Yaskawa INFORM job: FRONT_SEARCH_0ST-2_5040.JBI

/JOB
//NAME FRONT_SEARCH_0ST-2_5040
///FOLDERNAME 02-SKRZYNIE_JOBS
//POS
///NPOS 102,102,0,15,0,0
///TOOL 0
///POSTYPE PULSE
///PULSE
C00000=0,-52280,40443,0,-64237,0
C00001=0,-44333,40442,1,-36510,2
C00002=0,-77502,-19682,2,-20075,2
C00003=-31499,-58302,-23356,15027,12889,-13082
C00004=-52768,-43016,-26078,18373,38595,-18774
C00005=-77982,-19483,-4354,30116,56383,-30765
C00006=-53036,-11528,-12218,12363,64665,-17409
C00007=-53036,-11528,-12218,12363,64665,-17409
C00008=-51536,-9474,-10276,11905,64649,-16876
C00009=-51739,-9114,-7787,12104,63269,-17104
C00010=-53036,-11528,-12218,12363,64665,-17409
C00011=-17541,-26226,-24397,927,59032,-5038
C00012=-17541,-26226,-24397,927,59032,-5038
C00013=-16950,-23991,-22741,715,59568,-4818
C00014=-17036,-23563,-20101,755,58071,-4857
C00015=-17541,-26226,-24397,927,59032,-5038
C00016=34102,-23192,-21614,-15638,64271,13209
C00017=33423,-21885,-20599,-15423,64418,12942
C00018=32426,-19856,-18975,-15106,64629,12551
C00019=32578,-19611,-17013,-15290,63535,12762
C00020=33423,-21885,-20599,-15423,64418,12942
C00021=59339,-6070,-6417,-20979,72191,20891
C00022=59339,-6070,-6417,-20979,72191,20891
C00023=57897,-4256,-4562,-20702,71913,20431
C00024=58108,-3992,-2506,-20878,70835,20713
C00025=59339,-6070,-6417,-20979,72191,20891
C00026=42744,-35904,-30225,-18322,62562,16651
C00027=-53036,-11528,-12218,12363,64665,-17409
C00028=-77982,-26538,-29134,27151,66629,-27745
C00029=-70983,-8594,-1966,26503,59809,-49670
C00030=-80152,19776,40785,37351,72704,-50428
C00031=-79984,20154,42529,37516,71911,-50638
C00032=-79233,18397,40079,37458,71885,-50340
C00033=-79984,20154,42529,37516,71911,-50638
C00034=-73519,23289,38838,28890,77081,-45618
C00035=-73519,24511,42682,29072,75582,-46027
C00036=-73519,23289,38838,28890,77081,-45618
C00037=-88897,15706,42282,50101,71325,-56974
C00038=-88897,15706,42282,50101,71325,-56974
C00039=-87612,12343,37838,50071,70996,-56519
C00040=-85283,14202,40272,50301,69633,-56165
C00041=-87338,12550,38107,50098,70839,-56476
C00042=-84952,-1789,13569,34660,47724,-58955
C00043=-67641,-1674,11109,10330,44856,-44725
C00044=-66443,961,13975,9688,44721,-44210
C00045=-67641,-1674,11109,10330,44856,-44725
C00046=-67641,-376,15347,10694,42950,-44967
C00047=-67641,-1674,11109,10330,44856,-44725
C00048=-79040,417,20398,15965,28992,-57786
C00049=-76655,5212,30978,15501,25024,-57306
C00050=-76655,6949,35816,16758,23084,-57955
C00051=-76655,5212,30978,15501,25024,-57306
C00052=-74761,6919,33010,13466,24593,-56049
C00053=-80460,-2874,12270,15804,32253,-57809
C00054=-61258,-29124,-13156,26560,43617,-22150
C00055=-30420,-40507,-29240,27153,53235,15188
C00056=-18589,-38725,-21450,23338,47896,18931
C00057=-17722,-35233,-16455,23322,46926,19051
C00058=-17722,-33749,-12435,23948,45421,18620
C00059=-17722,-33892,-12819,23887,45564,18661
C00060=-16677,-31133,-11209,23138,46167,19311
C00061=-17819,-35820,-17540,23246,47228,19090
C00062=-74104,-11494,-6266,31916,75042,4269
C00063=-71226,-7329,2631,32115,71468,4273
C00064=-71226,-6504,5446,32343,70365,3922
C00065=-71226,-6611,5086,32313,70505,3967
C00066=-68386,-4058,7675,32040,69573,4789
C00067=-73314,-9412,-353,32206,72648,3829
C00068=51751,-31069,-22965,-10739,49070,48663
C00069=49028,-23852,-11575,-9841,46366,47823
C00070=49028,-23004,-8935,-10039,45204,47956
C00071=49028,-23118,-9286,-10013,45357,47939
C00072=47000,-20813,-7527,-8928,45644,47024
C00073=50476,-26208,-15307,-10408,47325,48332
C00074=90602,-5375,6902,-38786,69848,59444
C00075=83174,19950,50269,-44999,67580,58220
C00076=82362,17902,47383,-44926,67511,57879
C00077=83515,19072,48341,-44798,68200,58056
C00078=78091,19382,40247,-36371,72286,52960
C00079=78091,20664,44011,-36670,70997,53443
C00080=78091,19382,40247,-36371,72286,52960
C00081=88699,7296,38566,-55615,63182,60372
C00082=86803,3068,32674,-55410,62638,59657
C00083=84852,4315,34115,-55564,61561,59330
C00084=86803,3068,32674,-55410,62638,59657
C00085=92770,-2803,21719,-53893,67577,59421
C00086=73393,-10627,10934,-27897,30744,62458
C00087=70789,-6606,18800,-27824,27830,62140
C00088=69654,-4593,20814,-26755,27596,61444
C00089=70789,-6606,18800,-27824,27830,62140
C00090=70789,-5070,23059,-29482,26284,63017
C00091=70789,-6606,18800,-27824,27830,62140
C00092=83486,-8736,6503,-27040,35338,66550
C00093=77831,-2041,26192,-25270,18452,68895
C00094=77967,1961,32070,-26860,17569,69698
C00095=77967,5243,40752,-32914,14549,72656
C00096=77967,1961,32070,-26860,17569,69698
C00097=74560,4730,35257,-21622,16551,66717
C00098=77967,1961,32070,-26860,17569,69698
C00099=81109,-22356,2664,-22493,33121,60116
C00100=86168,-49730,-13668,-23926,46819,49343
C00101=44183,-52048,-7537,-24795,46064,51426
BC00000=868944
BC00001=857186
BC00002=897097
BC00003=897097
BC00004=897097
BC00005=897097
BC00006=912458
BC00007=912458
BC00008=912458
BC00009=912458
BC00010=912458
BC00011=912458
BC00012=912458
BC00013=912458
BC00014=912458
BC00015=912458
BC00016=912458
BC00017=912458
BC00018=912458
BC00019=912458
BC00020=912458
BC00021=912458
BC00022=912458
BC00023=912458
BC00024=912458
BC00025=912458
BC00026=912458
BC00027=912458
BC00028=912458
BC00029=912458
BC00030=912458
BC00031=912460
BC00032=912460
BC00033=912460
BC00034=912460
BC00035=912460
BC00036=912460
BC00037=912460
BC00038=912460
BC00039=912460
BC00040=912460
BC00041=912460
BC00042=912460
BC00043=912460
BC00044=912460
BC00045=912460
BC00046=912460
BC00047=912460
BC00048=912460
BC00049=912460
BC00050=912460
BC00051=912460
BC00052=912460
BC00053=912460
BC00054=912461
BC00055=912462
BC00056=912462
BC00057=912462
BC00058=912462
BC00059=912462
BC00060=912462
BC00061=912462
BC00062=912462
BC00063=912462
BC00064=912462
BC00065=912462
BC00066=912434
BC00067=912448
BC00068=912448
BC00069=912448
BC00070=912448
BC00071=912448
BC00072=912448
BC00073=912448
BC00074=912462
BC00075=912462
BC00076=912462
BC00077=912462
BC00078=912462
BC00079=912462
BC00080=912462
BC00081=912462
BC00082=912462
BC00083=912462
BC00084=912462
BC00085=912462
BC00086=912462
BC00087=912462
BC00088=912462
BC00089=912462
BC00090=912462
BC00091=912462
BC00092=912462
BC00093=912462
BC00094=912462
BC00095=912462
BC00096=912462
BC00097=912462
BC00098=912462
BC00099=880677
BC00100=854232
BC00101=807451
///POSTYPE BASE
///RECTAN
///RCONF 1,0,0,0,0,0,0,0,0,0,0,0,0,0,0,0,0,0,0,0,0,0,0,0
P00006=0.000,0.000,0.000,0.0000,0.0000,0.0000
///RCONF 0,0,0,0,0,0,0,0,0,0,0,0,0,0,0,0,0,0,0,0,0,0,0,0
P00058=0.000,0.000,3.000,0.0000,0.0000,0.0000
P00350=11.519,-0.008,1.149,0.0000,0.0000,0.0000
P00351=13.563,-0.027,-0.653,0.0000,0.0000,0.0000
P00352=13.252,-0.027,-0.827,0.0000,0.0000,0.0000
P00353=10.971,-0.082,0.776,0.0000,0.0000,0.0000
P00399=-2.449,0.031,8.825,0.0000,0.0000,0.0000
P00400=5.920,-3.503,-0.024,0.0000,0.0000,0.0000
P00401=3.430,-0.021,1.131,0.0000,0.0000,0.0000
P00402=-0.253,1.107,3.062,0.0000,0.0000,0.0000
P00403=-3.666,-0.015,5.328,0.0000,0.0000,0.0000
P00405=2.420,0.007,1.427,0.0000,0.0000,0.0000
P00406=3.513,-0.022,0.429,0.0000,0.0000,0.0000
P00415=-1.781,-1.303,3.250,0.0000,0.0000,0.0000
P00416=0.027,1.119,3.078,0.0000,0.0000,0.0000
//INST
///DATE 2024/05/14 19:22
///ATTR SC,RW
///GROUP1 RB1,BS1
NOP
MOVJ C00000 BC00000 VJ=10.00
MOVJ C00001 BC00001 VJ=30.00
MOVJ C00002 BC00002 VJ=20.00
MOVJ C00003 BC00003 VJ=20.00
MOVJ C00004 BC00004 VJ=20.00
MOVJ C00005 BC00005 VJ=10.00
'DODANE
'SZUKANIE FRONT
'------------------------
'503
'------------------------
MOVL C00006 BC00006 V=166.7
MOVL C00007 BC00007 V=66.7 PL=0
REFP 3 C00008 BC00008
CALL JOB:SEARCH-R1
IMOV P0058 V=16.7
SET P0350 P0006
SFTON P0350
REFP 3 C00009 BC00009
CALL JOB:SEARCH-R1
SET P0350 P0006
SFTON P0350
MOVL C00010 BC00010 V=66.7 PL=0
SFTOF
'------------------------
'------------------------
'502
'------------------------
MOVL C00011 BC00011 V=166.7
MOVL C00012 BC00012 V=66.7 PL=0
REFP 3 C00013 BC00013
CALL JOB:SEARCH-R1
IMOV P0058 V=16.7
SET P0351 P0006
SFTON P0351
REFP 3 C00014 BC00014
CALL JOB:SEARCH-R1
SET P0351 P0006
SFTON P0351
MOVL C00015 BC00015 V=66.7 PL=0
SFTOF
'------------------------
'------------------------
'501
'------------------------
MOVL C00016 BC00016 V=166.7
MOVL C00017 BC00017 V=66.7 PL=0
REFP 3 C00018 BC00018
CALL JOB:SEARCH-R1
IMOV P0058 V=16.7
SET P0352 P0006
SFTON P0352
REFP 3 C00019 BC00019
CALL JOB:SEARCH-R1
SET P0352 P0006
SFTON P0352
MOVL C00020 BC00020 V=66.7 PL=0
SFTOF
'------------------------
'------------------------
'500
'------------------------
MOVL C00021 BC00021 V=166.7
MOVL C00022 BC00022 V=66.7 PL=0
REFP 3 C00023 BC00023
CALL JOB:SEARCH-R1
IMOV P0058 V=16.7
SET P0353 P0006
SFTON P0353
REFP 3 C00024 BC00024
CALL JOB:SEARCH-R1
SET P0353 P0006
SFTON P0353
MOVL C00025 BC00025 V=66.7 PL=0
SFTOF
'------------------------
MOVL C00026 BC00026 V=333.3
MOVL C00027 BC00027 V=333.3
MOVJ C00028 BC00028 VJ=10.00
'DODANE
MOVJ C00029 BC00029 VJ=10.00
'------------------------
'SFT402
'------------------------
SFTOF
MOVL C00030 BC00030 V=150.0
MOVL C00031 BC00031 V=66.7 PL=0
REFP 3 C00032 BC00032
CALL JOB:SEARCH-R1
SET P0402 P0006
SFTON P0402
MOVL C00033 BC00033 V=150.0
MOVL C00034 BC00034 V=66.7 PL=0
REFP 3 C00035 BC00035
CALL JOB:SEARCH-R1
SET P0402 P0006
SFTON P0402
MOVL C00036 BC00036 V=133.3
MOVL C00037 BC00037 V=150.0
MOVL C00038 BC00038 V=150.0
MOVL C00039 BC00039 V=66.7 PL=0
REFP 3 C00040 BC00040
CALL JOB:SEARCH-R1
SET P0402 P0006
SFTOF
MOVL C00041 BC00041 V=150.0
'------------------------
'SFT403
'------------------------
'START
SFTOF
MOVL C00042 BC00042 V=250.0
MOVL C00043 BC00043 V=133.3 PL=0
REFP 3 C00044 BC00044
CALL JOB:SEARCH-R1
SET P0416 P0006
SFTON P0416
MOVL C00045 BC00045 V=133.3
REFP 3 C00046 BC00046
CALL JOB:SEARCH-R1
SET P0402 P0006
SFTOF
MOVL C00047 BC00047 V=150.0
'------------------------
'------------------------
SFTOF
MOVL C00048 BC00048 V=250.0
MOVL C00049 BC00049 V=133.3 PL=0
REFP 3 C00050 BC00050
CALL JOB:SEARCH-R1
SET P0403 P0006
SFTON P0403
MOVL C00051 BC00051 V=66.7 PL=0
REFP 3 C00052 BC00052
CALL JOB:SEARCH-R1
SET P0403 P0006
SFTOF
MOVL C00053 BC00053 V=150.0
MOVJ C00054 BC00054 VJ=20.00
MOVJ C00055 BC00055 VJ=20.00
'------------------------
'SFT401
'------------------------
SFTOF
MOVL C00056 BC00056 V=150.0
MOVL C00057 BC00057 V=66.7 PL=0
REFP 3 C00058 BC00058
CALL JOB:SEARCH-R1
SET P0401 P0006
SFTON P0401
MOVL C00059 BC00059 V=66.7 PL=0
REFP 3 C00060 BC00060
CALL JOB:SEARCH-R1
SET P0401 P0006
SFTOF
MOVL C00061 BC00061 V=150.0
'SFT400
'------------------------
SFTOF
MOVL C00062 BC00062 V=333.3
MOVL C00063 BC00063 V=66.7 PL=0
REFP 3 C00064 BC00064
CALL JOB:SEARCH-R1
SET P0405 P0006
SFTON P0405
MOVL C00065 BC00065 V=66.7 PL=0
REFP 3 C00066 BC00066
CALL JOB:SEARCH-R1
SET P0405 P0006
SFTOF
MOVL C00067 BC00067 V=150.0
'SFT400
'------------------------
SFTOF
MOVL C00068 BC00068 V=333.3
MOVL C00069 BC00069 V=133.3 PL=0
REFP 3 C00070 BC00070
CALL JOB:SEARCH-R1
SET P0406 P0006
SFTON P0406
MOVL C00071 BC00071 V=66.7 PL=0
REFP 3 C00072 BC00072
CALL JOB:SEARCH-R1
SET P0406 P0006
SFTOF
MOVL C00073 BC00073 V=150.0
'SFT400
'------------------------
SFTOF
MOVL C00074 BC00074 V=150.0
MOVL C00075 BC00075 V=66.7 PL=0
REFP 3 C00076 BC00076
CALL JOB:SEARCH-R1
SET P0400 P0006
SFTON P0400
MOVL C00077 BC00077 V=150.0
MOVL C00078 BC00078 V=66.7 PL=0
REFP 3 C00079 BC00079
CALL JOB:SEARCH-R1
SET P0400 P0006
SFTON P0400
MOVL C00080 BC00080 V=150.0
MOVL C00081 BC00081 V=150.0
MOVL C00082 BC00082 V=66.7 PL=0
REFP 3 C00083 BC00083
CALL JOB:SEARCH-R1
SET P0400 P0006
SFTOF
MOVL C00084 BC00084 V=83.3
MOVL C00085 BC00085 V=250.0
MOVL C00086 BC00086 V=333.3
MOVL C00087 BC00087 V=66.7 PL=0
REFP 3 C00088 BC00088
CALL JOB:SEARCH-R1
SET P0415 P0006
SFTON P0415
MOVL C00089 BC00089 V=133.3
REFP 3 C00090 BC00090
CALL JOB:SEARCH-R1
SET P0415 P0006
SFTOF
MOVL C00091 BC00091 V=150.0
'------------------------
'SFT403
'------------------------
'START
SFTOF
MOVJ C00092 BC00092 VJ=10.00
'------------------------
'SFT399
'------------------------
'START
SFTOF
MOVL C00093 BC00093 V=150.0
MOVL C00094 BC00094 V=66.7 PL=0
REFP 3 C00095 BC00095
CALL JOB:SEARCH-R1
SET P0399 P0006
SFTON P0399
MOVL C00096 BC00096 V=66.7 PL=0
REFP 3 C00097 BC00097
CALL JOB:SEARCH-R1
SET P0399 P0006
SFTOF
MOVL C00098 BC00098 V=150.0
MOVJ C00099 BC00099 VJ=20.00
MOVJ C00100 BC00100 VJ=30.00
MOVJ C00101 BC00101 VJ=30.00
END
